{attribute 'GeneratedUsingTerminal: EK1100-0000-0018'}
{attribute addProperty BoxType "EK1100-0000-0018"}
{attribute addProperty Id "Beckhoff_EP4xxxEK1122Beckhoff_EP4xxxEK1122_1E5F5BC9336"}
{attribute addProperty CRC "2145098522"}
{attribute addProperty Size "336"}
TYPE Beckhoff_EP4xxx_7FDB9B1A EXTENDS EK1100_1FC0878B :
STRUCT
	{attribute addProperty Name "Beckhoff_EP4xxxEK1122"}
	{attribute addProperty PreviousPort "Beckhoff EP4xxx : B"}
	Beckhoff_EP4xxxEK1122 : Beckhoff_EP4xxxEK1122_1E5F5BC9;
END_STRUCT
END_TYPE

(* stored: Version 1.2.0.0, ProductVersion 3.1.4024.9
   DUT Beckhoff_EP4xxx_7FDB9B1A: Id {64b5e2b3-5372-4fa1-a2d3-8ae9a1b1bcf9} *)
